// Mitsubishi GX Works2 project: PLC   PLC: Q03UD

PROGRAM MAIN
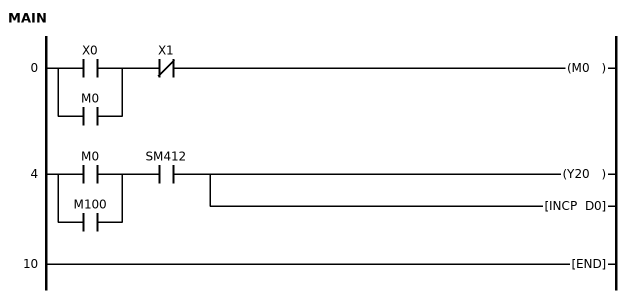
0     LD      X0
      OR      M0
      ANI     X1
      OUT     M0
4     LD      M0
      OR      M100
      AND     SM412
      OUT     Y20
      INCP    D0
10    END
END_PROGRAM
